# EPICS autosave request: BPMApp/Db/BPMAdc_settings.req
$(P)$(R)ADCSw
$(P)$(R)ADCSwDly
$(P)$(R)ADCSwDivClk
$(P)$(R)ADCTrigDir
$(P)$(R)ADCTrigTerm
$(P)$(R)ADCSi57xFreq
$(P)$(R)ADCAD9510PllFunc
$(P)$(R)ADCAD9510ClkSel
$(P)$(R)ADCAD9510ADiv
$(P)$(R)ADCAD9510BDiv
$(P)$(R)ADCAD9510Prescaler
$(P)$(R)ADCAD9510RDiv
$(P)$(R)ADCAD9510PllPDown
$(P)$(R)ADCAD9510MuxStatus
$(P)$(R)ADCAD9510CpCurrent
$(P)$(R)ADCAD9510Outputs
